FUNCTION_BLOCK GET_PLANE_EQUATION
  (* Standard: 61499-2 *)
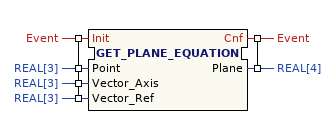
  EVENT_INPUT
    Init WITH Point, Vector_Axis, Vector_Ref;
  END_EVENT
  EVENT_OUTPUT
    Cnf WITH Plane;
  END_EVENT
  VAR_INPUT
    Point : ARRAY [0..2] OF REAL;
    Vector_Axis : ARRAY [0..2] OF REAL;
    Vector_Ref : ARRAY [0..2] OF REAL;
  END_VAR
  VAR_OUTPUT
    Plane : ARRAY [0..3] OF REAL;
  END_VAR
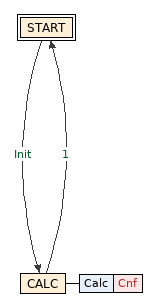
  EC_STATES
    START;
    CALC : Calc -> Cnf;
  END_STATES
  EC_TRANSITIONS
    START TO CALC := Init;
    CALC TO START := 1;
  END_TRANSITIONS
  ALGORITHM Calc IN Lua:
    if Vector_Axis == '$' or Vector_Ref == '$' or not Vector_Axis or not Vector_Ref
	or (Vector_Axis[1] == 0 and Vector_Axis[2] == 0 and Vector_Axis[3] ==0 ) then
	Plane = {0, 0, 1, Point[3]}
else
	local normal = Vector_Axis
	local m	     = sqrt (normal[1]^2 + normal[2]^2 + normal[3]^2)
	normal = {
		normal[1]/m,
		normal[2]/m,
		normal[3]/m
	}
	local p = Point
	print('GET_PLANE Point', Point[1], Point[2], Point[3])
	Plane   = {normal[1], normal[2], normal[3], p[1]*normal[1] + p[2]*normal[2] + p[3]*normal[3]}
end
	print('GET_PLANE Vector_Axis', Vector_Axis[1], Vector_Axis[2], Vector_Axis[3])
	print('GET_PLANE Plane', Plane[1], Plane[2], Plane[3], Plane[4])
  END_ALGORITHM
END_FUNCTION_BLOCK
